ABB RobotStudio station: ABB_Project_EGM_Stream_Single.rspag

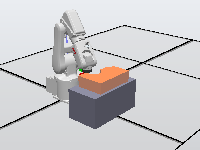
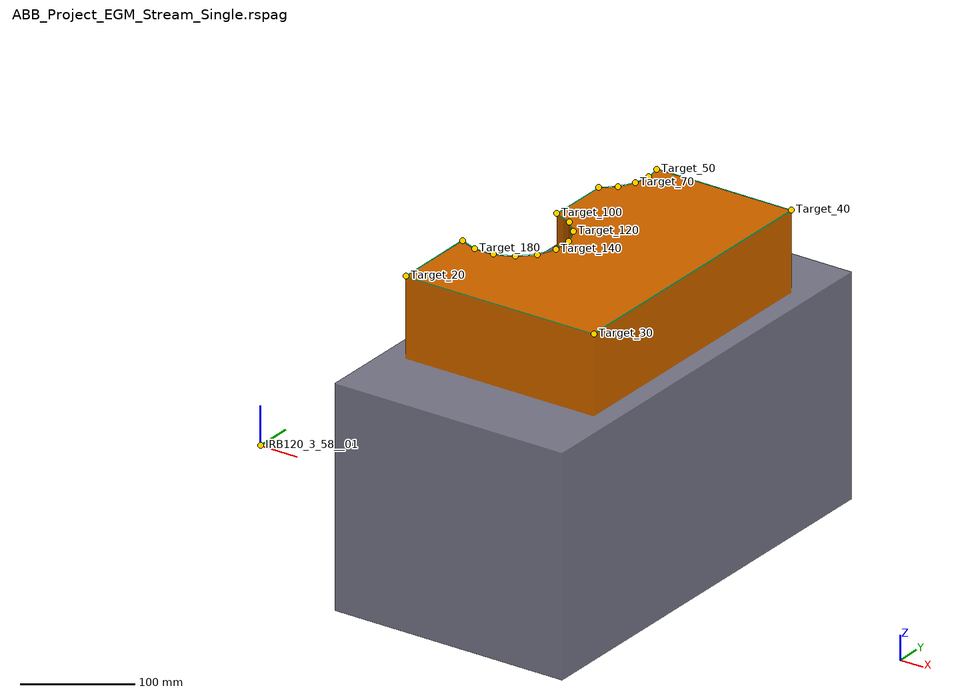
[picture v1: parts stored in the station drawn from their meshes, with robot base, taught points and paths (robot models come from the ABB library and are not in the file)]
--- station ---
Station ABB_Project_EGM_Control (saved by RobotStudio 21.2.9526.0)
Controller Controller2
  mechanical unit ROB_1: IRB120_3_58__01, 6 joints, base frame (0, 0, 0) mm
Layout (positions relative to the parent item):
  - Pad [part] at (250, 150, 200) mm, rotated rx 0 ry 0 rz -90 deg, size 300 x 200 x 100 mm
  - Table [part] at (-40, 0, 0) mm, size 242 x 440 x 220 mm
  - IRB120_3_58__01 [mechanism, from Robots\IRB120_3_58_G_01.rslib] at (0, 0, 0) mm; joint values [-0.2562, 0.0921, 0.7826, 0, 0.6961, -1.827] (rad or m)
Targets, tools, work objects and paths stored in the station and not in the controller backup, written as RAPID:
! task T_ROB1
MODULE Module1
  CONST robtarget Target_10_2:=[[263.321960449,-68.978512397,300],[0,-0.707106781,0.707106781,0],[-1,0,-2,0],[9E+09,9E+09,9E+09,9E+09,9E+09,9E+09]];
  CONST robtarget Target_20_3:=[[263.321960449,-155.446746826,300],[0,-0.707106781,0.707106781,0],[-1,0,-2,0],[9E+09,9E+09,9E+09,9E+09,9E+09,9E+09]];
  CONST robtarget Target_30_3:=[[463.321960449,-155.446746826,300],[0,-0.707106781,0.707106781,0],[-1,0,-2,0],[9E+09,9E+09,9E+09,9E+09,9E+09,9E+09]];
  CONST robtarget Target_40_3:=[[463.321960449,144.553253174,300],[0,-0.707106781,0.707106781,0],[0,0,-1,0],[9E+09,9E+09,9E+09,9E+09,9E+09,9E+09]];
  CONST robtarget Target_50_3:=[[320.448416208,144.553253174,300],[0,-0.707106781,0.707106781,0],[0,0,-1,0],[9E+09,9E+09,9E+09,9E+09,9E+09,9E+09]];
  CONST robtarget Target_60_3:=[[323.349310221,127.995106698,300],[0,-0.707106781,0.707106781,0],[0,0,-1,0],[9E+09,9E+09,9E+09,9E+09,9E+09,9E+09]];
  CONST robtarget Target_70_3:=[[320.59851418,111.411363998,300],[0,-0.707106781,0.707106781,0],[0,0,-1,0],[9E+09,9E+09,9E+09,9E+09,9E+09,9E+09]];
  CONST robtarget Target_80_3:=[[312.506964207,96.676567771,300],[0,-0.707106781,0.707106781,0],[0,0,-1,0],[9E+09,9E+09,9E+09,9E+09,9E+09,9E+09]];
  CONST robtarget Target_90_3:=[[299.98928833,85.456265126,300],[0,-0.707106781,0.707106781,0],[0,0,-1,0],[9E+09,9E+09,9E+09,9E+09,9E+09,9E+09]];
  CONST robtarget Target_100_3:=[[299.98928833,22.036067079,300],[0,-0.707106781,0.707106781,0],[0,0,-1,0],[9E+09,9E+09,9E+09,9E+09,9E+09,9E+09]];
  CONST robtarget Target_110_3:=[[318.046831052,14.718242482,300],[0,-0.707106781,0.707106781,0],[0,0,-1,0],[9E+09,9E+09,9E+09,9E+09,9E+09,9E+09]];
  CONST robtarget Target_120_3:=[[331.936397486,1.05422586,300],[0,-0.707106781,0.707106781,0],[0,0,-1,0],[9E+09,9E+09,9E+09,9E+09,9E+09,9E+09]];
  CONST robtarget Target_130_3:=[[339.548854715,-16.881099643,300],[0,-0.707106781,0.707106781,0],[-1,0,-2,0],[9E+09,9E+09,9E+09,9E+09,9E+09,9E+09]];
  CONST robtarget Target_140_3:=[[339.728249872,-36.364251938,300],[0,-0.707106781,0.707106781,0],[-1,0,-2,0],[9E+09,9E+09,9E+09,9E+09,9E+09,9E+09]];
  CONST robtarget Target_150_3:=[[332.447341773,-54.436711185,300],[0,-0.707106781,0.707106781,0],[-1,0,-2,0],[9E+09,9E+09,9E+09,9E+09,9E+09,9E+09]];
  CONST robtarget Target_160_3:=[[318.811737495,-68.354171512,300],[0,-0.707106781,0.707106781,0],[-1,0,-2,0],[9E+09,9E+09,9E+09,9E+09,9E+09,9E+09]];
  CONST robtarget Target_170_3:=[[300.892005763,-76.003264309,300],[0,-0.707106781,0.707106781,0],[-1,0,-2,0],[9E+09,9E+09,9E+09,9E+09,9E+09,9E+09]];
  CONST robtarget Target_180_3:=[[281.40926075,-76.222473592,300],[0,-0.707106781,0.707106781,0],[-1,0,-2,0],[9E+09,9E+09,9E+09,9E+09,9E+09,9E+09]];
  CONST robtarget Target_190_3:=[[263.321960449,-68.978512397,300],[0,-0.707106781,0.707106781,0],[-1,0,-2,0],[9E+09,9E+09,9E+09,9E+09,9E+09,9E+09]];
  CONST robtarget Target_20_2_3:=[[263.321960449,-155.446746826,300],[0,-0.382683433,0.923879532,0],[-1,0,-1,0],[9E+09,9E+09,9E+09,9E+09,9E+09,9E+09]];
  CONST robtarget Target_30_2_3:=[[463.321960449,-155.446746826,300],[0,0.923879532,-0.382683433,0],[-1,0,-2,0],[9E+09,9E+09,9E+09,9E+09,9E+09,9E+09]];
  CONST robtarget Target_40_2_3:=[[463.321960449,144.553253174,300],[0,0.923879533,0.382683431,0],[0,0,-3,0],[9E+09,9E+09,9E+09,9E+09,9E+09,9E+09]];
  CONST robtarget Target_50_2_3:=[[320.448416208,144.553253174,300],[0,-0.608761429,0.79335334,0],[0,0,-1,0],[9E+09,9E+09,9E+09,9E+09,9E+09,9E+09]];
  CONST robtarget Target_60_2_3:=[[323.349310221,127.995106698,300],[0,-0.5,0.866025404,0],[0,0,-1,0],[9E+09,9E+09,9E+09,9E+09,9E+09,9E+09]];
  CONST robtarget Target_70_2_3:=[[320.59851418,111.411363998,300],[0,-0.382683432,0.923879533,0],[0,0,-1,0],[9E+09,9E+09,9E+09,9E+09,9E+09,9E+09]];
  CONST robtarget Target_80_2_3:=[[312.506964207,96.676567771,300],[0,-0.258819045,0.965925826,0],[0,0,-1,0],[9E+09,9E+09,9E+09,9E+09,9E+09,9E+09]];
  CONST robtarget Target_90_2_3:=[[299.98928833,85.456265126,300],[0,-0.130526192,0.991444861,0],[0,0,0,0],[9E+09,9E+09,9E+09,9E+09,9E+09,9E+09]];
  CONST robtarget Target_100_2_3:=[[299.98928833,22.036067079,300],[0,0.923879533,0.382683432,0],[0,0,1,0],[9E+09,9E+09,9E+09,9E+09,9E+09,9E+09]];
  CONST robtarget Target_110_2_3:=[[318.046831052,14.718242482,300],[0,0.965925826,0.258819045,0],[0,0,1,0],[9E+09,9E+09,9E+09,9E+09,9E+09,9E+09]];
  CONST robtarget Target_120_2_3:=[[331.936397486,1.05422586,300],[0,0.991444861,0.130526192,0],[0,0,1,0],[9E+09,9E+09,9E+09,9E+09,9E+09,9E+09]];
  CONST robtarget Target_130_2_3:=[[339.548854715,-16.881099643,300],[0,1,0,0],[-1,0,1,0],[9E+09,9E+09,9E+09,9E+09,9E+09,9E+09]];
  CONST robtarget Target_140_2_3:=[[339.728249872,-36.364251938,300],[0,0.991444861,-0.130526192,0],[-1,0,2,0],[9E+09,9E+09,9E+09,9E+09,9E+09,9E+09]];
  CONST robtarget Target_150_2_3:=[[332.447341773,-54.436711185,300],[0,0.965925826,-0.258819045,0],[-1,0,2,0],[9E+09,9E+09,9E+09,9E+09,9E+09,9E+09]];
  CONST robtarget Target_160_2_3:=[[318.811737495,-68.354171512,300],[0,0.923879533,-0.382683432,0],[-1,0,2,0],[9E+09,9E+09,9E+09,9E+09,9E+09,9E+09]];
  CONST robtarget Target_170_2_3:=[[300.892005763,-76.003264309,300],[0,0.866025404,-0.5,0],[-1,0,2,0],[9E+09,9E+09,9E+09,9E+09,9E+09,9E+09]];
  CONST robtarget Target_180_2_3:=[[281.40926075,-76.222473592,300],[0,0.79335334,-0.608761429,0],[-1,0,2,0],[9E+09,9E+09,9E+09,9E+09,9E+09,9E+09]];
  CONST robtarget Target_190_2_4:=[[263.321960449,-68.978512397,300],[0,-0.707106781,0.707106781,0],[-1,0,2,0],[9E+09,9E+09,9E+09,9E+09,9E+09,9E+09]];
  CONST robtarget Target_10_2_2_2:=[[263.321960449,-68.978512397,300],[0.092295956,-0.701057385,0.701057385,-0.092295956],[-1,0,-2,0],[9E+09,9E+09,9E+09,9E+09,9E+09,9E+09]];
  CONST robtarget Target_20_2_2_3:=[[263.321960449,-155.446746826,300],[0.092295956,-0.701057385,0.701057385,-0.092295956],[-1,0,-2,0],[9E+09,9E+09,9E+09,9E+09,9E+09,9E+09]];
  CONST robtarget Target_20_2_2_2_2:=[[263.321960449,-155.446746826,300],[0,-0.382683433,0.923879532,0],[-1,0,-1,0],[9E+09,9E+09,9E+09,9E+09,9E+09,9E+09]];
  CONST robtarget Target_30_2_2_3:=[[463.321960449,-155.446746826,300],[0,0.923879532,-0.382683433,0],[-1,0,-2,0],[9E+09,9E+09,9E+09,9E+09,9E+09,9E+09]];
  CONST robtarget Target_30_2_2_2_2:=[[463.321960449,-155.446746826,300],[0.037109679,0.916827972,-0.387892623,-0.087112884],[-1,-1,-2,0],[9E+09,9E+09,9E+09,9E+09,9E+09,9E+09]];
  CONST robtarget Target_40_2_2_3:=[[463.321960449,144.553253174,300],[0.037109679,0.916827972,-0.387892623,-0.087112884],[0,0,-2,0],[9E+09,9E+09,9E+09,9E+09,9E+09,9E+09]];
  CONST robtarget Target_40_2_2_2_2:=[[463.321960449,144.553253174,300],[0,0.923879533,0.382683431,0],[0,0,-3,0],[9E+09,9E+09,9E+09,9E+09,9E+09,9E+09]];
  CONST robtarget Target_60_2_2_2:=[[323.349310221,127.995106698,300],[0,-0.5,0.866025404,0],[0,0,-1,0],[9E+09,9E+09,9E+09,9E+09,9E+09,9E+09]];
  CONST robtarget Target_70_2_2_2:=[[320.59851418,111.411363998,300],[0,-0.382683432,0.923879533,0],[0,0,-1,0],[9E+09,9E+09,9E+09,9E+09,9E+09,9E+09]];
  CONST robtarget Target_80_2_2_2:=[[312.506964207,96.676567771,300],[0,-0.258819045,0.965925826,0],[0,0,-1,0],[9E+09,9E+09,9E+09,9E+09,9E+09,9E+09]];
  CONST robtarget Target_90_2_2_2:=[[299.98928833,85.456265126,300],[0,-0.130526192,0.991444861,0],[0,0,0,0],[9E+09,9E+09,9E+09,9E+09,9E+09,9E+09]];
  CONST robtarget Target_100_2_2_2:=[[299.98928833,22.036067079,300],[0,0.923879533,0.382683432,0],[0,0,1,0],[9E+09,9E+09,9E+09,9E+09,9E+09,9E+09]];
  CONST robtarget Target_110_2_2_2:=[[318.046831052,14.718242482,300],[0,0.965925826,0.258819045,0],[0,0,1,0],[9E+09,9E+09,9E+09,9E+09,9E+09,9E+09]];
  CONST robtarget Target_120_2_2_2:=[[331.936397486,1.05422586,300],[0,0.991444861,0.130526192,0],[0,0,1,0],[9E+09,9E+09,9E+09,9E+09,9E+09,9E+09]];
  CONST robtarget Target_130_2_2_2:=[[339.548854715,-16.881099643,300],[0,1,0,0],[-1,0,1,0],[9E+09,9E+09,9E+09,9E+09,9E+09,9E+09]];
  CONST robtarget Target_140_2_2_2:=[[339.728249872,-36.364251938,300],[0,0.991444861,-0.130526192,0],[-1,0,2,0],[9E+09,9E+09,9E+09,9E+09,9E+09,9E+09]];
  CONST robtarget Target_150_2_2_2:=[[332.447341773,-54.436711185,300],[0,0.965925826,-0.258819045,0],[-1,0,2,0],[9E+09,9E+09,9E+09,9E+09,9E+09,9E+09]];
  CONST robtarget Target_160_2_2_2:=[[318.811737495,-68.354171512,300],[0,0.923879533,-0.382683432,0],[-1,0,2,0],[9E+09,9E+09,9E+09,9E+09,9E+09,9E+09]];
  CONST robtarget Target_170_2_2_2:=[[300.892005763,-76.003264309,300],[0,0.866025404,-0.5,0],[-1,0,2,0],[9E+09,9E+09,9E+09,9E+09,9E+09,9E+09]];
  CONST robtarget Target_180_2_2_2:=[[281.40926075,-76.222473592,300],[0,0.79335334,-0.608761429,0],[-1,0,2,0],[9E+09,9E+09,9E+09,9E+09,9E+09,9E+09]];
  CONST robtarget Target_190_2_3_2:=[[263.321960449,-68.978512397,300],[0,-0.707106781,0.707106781,0],[-1,0,2,0],[9E+09,9E+09,9E+09,9E+09,9E+09,9E+09]];
  PROC Path_Experiment_1_T1()
    MoveL Target_10_2,v40,fine,tool0\WObj:=wobj0;
    MoveL Target_20_3,v40,fine,tool0\WObj:=wobj0;
    MoveL Target_30_3,v40,fine,tool0\WObj:=wobj0;
    MoveL Target_40_3,v40,fine,tool0\WObj:=wobj0;
    MoveL Target_50_3,v40,fine,tool0\WObj:=wobj0;
    MoveL Target_60_3,v40,fine,tool0\WObj:=wobj0;
    MoveL Target_70_3,v40,fine,tool0\WObj:=wobj0;
    MoveL Target_80_3,v40,fine,tool0\WObj:=wobj0;
    MoveL Target_90_3,v40,fine,tool0\WObj:=wobj0;
    MoveL Target_100_3,v40,fine,tool0\WObj:=wobj0;
    MoveL Target_110_3,v40,fine,tool0\WObj:=wobj0;
    MoveL Target_120_3,v40,fine,tool0\WObj:=wobj0;
    MoveL Target_130_3,v40,fine,tool0\WObj:=wobj0;
    MoveL Target_140_3,v40,fine,tool0\WObj:=wobj0;
    MoveL Target_150_3,v40,fine,tool0\WObj:=wobj0;
    MoveL Target_160_3,v40,fine,tool0\WObj:=wobj0;
    MoveL Target_170_3,v40,fine,tool0\WObj:=wobj0;
    MoveL Target_180_3,v40,fine,tool0\WObj:=wobj0;
    MoveL Target_190_3,v40,fine,tool0\WObj:=wobj0;
  ENDPROC
  PROC Path_Experiment_1_T2()
    MoveL Target_10_2,v40,fine,tool0\WObj:=wobj0;
    MoveL Target_20_2_3,v40,fine,tool0\WObj:=wobj0;
    MoveL Target_30_2_3,v40,fine,tool0\WObj:=wobj0;
    MoveL Target_40_2_3,v40,fine,tool0\WObj:=wobj0;
    MoveL Target_50_2_3,v40,fine,tool0\WObj:=wobj0;
    MoveL Target_60_2_3,v40,fine,tool0\WObj:=wobj0;
    MoveL Target_70_2_3,v40,fine,tool0\WObj:=wobj0;
    MoveL Target_80_2_3,v40,fine,tool0\WObj:=wobj0;
    MoveL Target_90_2_3,v40,fine,tool0\WObj:=wobj0;
    MoveL Target_100_2_3,v40,fine,tool0\WObj:=wobj0;
    MoveL Target_110_2_3,v40,fine,tool0\WObj:=wobj0;
    MoveL Target_120_2_3,v40,fine,tool0\WObj:=wobj0;
    MoveL Target_130_2_3,v40,fine,tool0\WObj:=wobj0;
    MoveL Target_140_2_3,v40,fine,tool0\WObj:=wobj0;
    MoveL Target_150_2_3,v40,fine,tool0\WObj:=wobj0;
    MoveL Target_160_2_3,v40,fine,tool0\WObj:=wobj0;
    MoveL Target_170_2_3,v40,fine,tool0\WObj:=wobj0;
    MoveL Target_180_2_3,v40,fine,tool0\WObj:=wobj0;
    MoveL Target_190_2_4,v40,fine,tool0\WObj:=wobj0;
  ENDPROC
  PROC Path_Experiment_1_T3()
    MoveL Target_10_2,v40,z10,tool0\WObj:=wobj0;
    MoveL Target_10_2_2_2,v40,z10,tool0\WObj:=wobj0;
    MoveL Target_20_2_2_3,v40,z10,tool0\WObj:=wobj0;
    MoveL Target_20_2_2_2_2,v40,z10,tool0\WObj:=wobj0;
    MoveL Target_30_2_2_3,v40,z10,tool0\WObj:=wobj0;
    MoveL Target_30_2_2_2_2,v40,z10,tool0\WObj:=wobj0;
    MoveL Target_40_2_2_3,v40,z10,tool0\WObj:=wobj0;
    MoveL Target_40_2_2_2_2,v40,z10,tool0\WObj:=wobj0;
    MoveL Target_50_2_2_2,v40,z10,tool0\WObj:=wobj0;
    MoveL Target_60_2_2_2,v40,z10,tool0\WObj:=wobj0;
    MoveL Target_70_2_2_2,v40,z10,tool0\WObj:=wobj0;
    MoveL Target_80_2_2_2,v40,z10,tool0\WObj:=wobj0;
    MoveL Target_90_2_2_2,v40,z10,tool0\WObj:=wobj0;
    MoveL Target_100_2_2_2,v40,z10,tool0\WObj:=wobj0;
    MoveL Target_110_2_2_2,v40,z10,tool0\WObj:=wobj0;
    MoveL Target_120_2_2_2,v40,z10,tool0\WObj:=wobj0;
    MoveL Target_130_2_2_2,v40,z10,tool0\WObj:=wobj0;
    MoveL Target_140_2_2_2,v40,z10,tool0\WObj:=wobj0;
    MoveL Target_150_2_2_2,v40,z10,tool0\WObj:=wobj0;
    MoveL Target_160_2_2_2,v40,z10,tool0\WObj:=wobj0;
    MoveL Target_170_2_2_2,v40,z10,tool0\WObj:=wobj0;
    MoveL Target_180_2_2_2,v40,z10,tool0\WObj:=wobj0;
    MoveL Target_190_2_3_2,v40,z10,tool0\WObj:=wobj0;
  ENDPROC
ENDMODULE


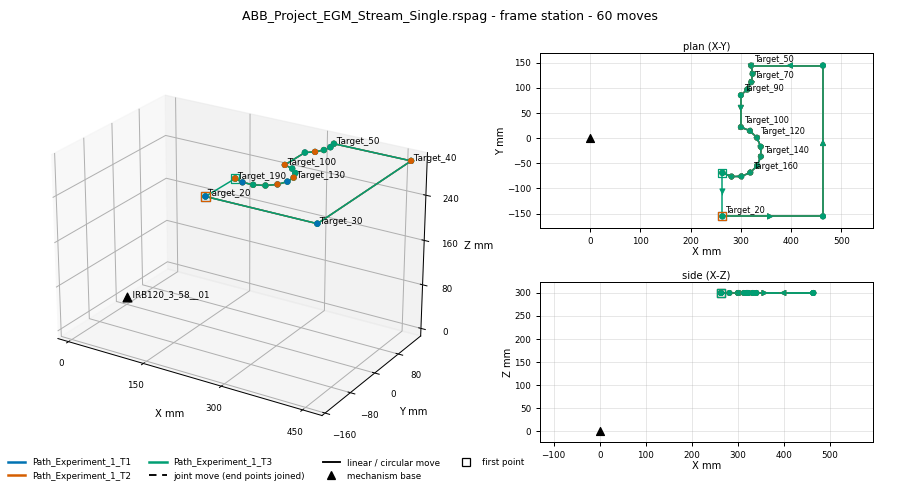
[picture p0: tool path of ABB_Project_EGM_Stream_Single.rspag in frame station, 60 of 60 moves have a stored position in this frame; points joined in program order, loops and branches not executed]
--- Backups/Controller2/RAPID/TASK1/PROGMOD/Module1.mod ---
MODULE Module1
    ! Targets
    CONST robtarget Target_10:=[[263.321960449,-68.978512397,300],[0,-0.707106781,0.707106781,0],[-1,0,-2,0],[9E+09,9E+09,9E+09,9E+09,9E+09,9E+09]];
    CONST robtarget Target_20:=[[263.321960449,-155.446746826,300],[0,-0.707106781,0.707106781,0],[-1,0,-2,0],[9E+09,9E+09,9E+09,9E+09,9E+09,9E+09]];
    CONST robtarget Target_30:=[[463.321960449,-155.446746826,300],[0,-0.707106781,0.707106781,0],[-1,0,-2,0],[9E+09,9E+09,9E+09,9E+09,9E+09,9E+09]];
    CONST robtarget Target_40:=[[463.321960449,144.553253174,300],[0,-0.707106781,0.707106781,0],[0,0,-1,0],[9E+09,9E+09,9E+09,9E+09,9E+09,9E+09]];
    CONST robtarget Target_50:=[[320.448416208,144.553253174,300],[0,-0.707106781,0.707106781,0],[0,0,-1,0],[9E+09,9E+09,9E+09,9E+09,9E+09,9E+09]];
    CONST robtarget Target_60:=[[323.349310221,127.995106698,300],[0,-0.707106781,0.707106781,0],[0,0,-1,0],[9E+09,9E+09,9E+09,9E+09,9E+09,9E+09]];
    CONST robtarget Target_70:=[[320.59851418,111.411363998,300],[0,-0.707106781,0.707106781,0],[0,0,-1,0],[9E+09,9E+09,9E+09,9E+09,9E+09,9E+09]];
    CONST robtarget Target_80:=[[312.506964207,96.676567771,300],[0,-0.707106781,0.707106781,0],[0,0,-1,0],[9E+09,9E+09,9E+09,9E+09,9E+09,9E+09]];
    CONST robtarget Target_90:=[[299.98928833,85.456265126,300],[0,-0.707106781,0.707106781,0],[0,0,-1,0],[9E+09,9E+09,9E+09,9E+09,9E+09,9E+09]];
    CONST robtarget Target_100:=[[299.98928833,22.036067079,300],[0,-0.707106781,0.707106781,0],[0,0,-1,0],[9E+09,9E+09,9E+09,9E+09,9E+09,9E+09]];
    CONST robtarget Target_110:=[[318.046831052,14.718242482,300],[0,-0.707106781,0.707106781,0],[0,0,-1,0],[9E+09,9E+09,9E+09,9E+09,9E+09,9E+09]];
    CONST robtarget Target_120:=[[331.936397486,1.05422586,300],[0,-0.707106781,0.707106781,0],[0,0,-1,0],[9E+09,9E+09,9E+09,9E+09,9E+09,9E+09]];
    CONST robtarget Target_130:=[[339.548854715,-16.881099643,300],[0,-0.707106781,0.707106781,0],[-1,0,-2,0],[9E+09,9E+09,9E+09,9E+09,9E+09,9E+09]];
    CONST robtarget Target_140:=[[339.728249872,-36.364251938,300],[0,-0.707106781,0.707106781,0],[-1,0,-2,0],[9E+09,9E+09,9E+09,9E+09,9E+09,9E+09]];
    CONST robtarget Target_150:=[[332.447341773,-54.436711185,300],[0,-0.707106781,0.707106781,0],[-1,0,-2,0],[9E+09,9E+09,9E+09,9E+09,9E+09,9E+09]];
    CONST robtarget Target_160:=[[318.811737495,-68.354171512,300],[0,-0.707106781,0.707106781,0],[-1,0,-2,0],[9E+09,9E+09,9E+09,9E+09,9E+09,9E+09]];
    CONST robtarget Target_170:=[[300.892005763,-76.003264309,300],[0,-0.707106781,0.707106781,0],[-1,0,-2,0],[9E+09,9E+09,9E+09,9E+09,9E+09,9E+09]];
    CONST robtarget Target_180:=[[281.40926075,-76.222473592,300],[0,-0.707106781,0.707106781,0],[-1,0,-2,0],[9E+09,9E+09,9E+09,9E+09,9E+09,9E+09]];
    CONST robtarget Target_190:=[[263.321960449,-68.978512397,300],[0,-0.707106781,0.707106781,0],[-1,0,-2,0],[9E+09,9E+09,9E+09,9E+09,9E+09,9E+09]];
    CONST robtarget Target_20_2:=[[263.321960449,-155.446746826,300],[0,-0.382683433,0.923879532,0],[-1,0,-1,0],[9E+09,9E+09,9E+09,9E+09,9E+09,9E+09]];
    CONST robtarget Target_30_2:=[[463.321960449,-155.446746826,300],[0,0.923879532,-0.382683433,0],[-1,0,-2,0],[9E+09,9E+09,9E+09,9E+09,9E+09,9E+09]];
    CONST robtarget Target_40_2:=[[463.321960449,144.553253174,300],[0,0.923879533,0.382683431,0],[0,0,-3,0],[9E+09,9E+09,9E+09,9E+09,9E+09,9E+09]];
    CONST robtarget Target_50_2:=[[320.448416208,144.553253174,300],[0,-0.608761429,0.79335334,0],[0,0,-1,0],[9E+09,9E+09,9E+09,9E+09,9E+09,9E+09]];
    CONST robtarget Target_60_2:=[[323.349310221,127.995106698,300],[0,-0.5,0.866025404,0],[0,0,-1,0],[9E+09,9E+09,9E+09,9E+09,9E+09,9E+09]];
    CONST robtarget Target_70_2:=[[320.59851418,111.411363998,300],[0,-0.382683432,0.923879533,0],[0,0,-1,0],[9E+09,9E+09,9E+09,9E+09,9E+09,9E+09]];
    CONST robtarget Target_80_2:=[[312.506964207,96.676567771,300],[0,-0.258819045,0.965925826,0],[0,0,-1,0],[9E+09,9E+09,9E+09,9E+09,9E+09,9E+09]];
    CONST robtarget Target_90_2:=[[299.98928833,85.456265126,300],[0,-0.130526192,0.991444861,0],[0,0,0,0],[9E+09,9E+09,9E+09,9E+09,9E+09,9E+09]];
    CONST robtarget Target_100_2:=[[299.98928833,22.036067079,300],[0,0.923879533,0.382683432,0],[0,0,1,0],[9E+09,9E+09,9E+09,9E+09,9E+09,9E+09]];
    CONST robtarget Target_110_2:=[[318.046831052,14.718242482,300],[0,0.965925826,0.258819045,0],[0,0,1,0],[9E+09,9E+09,9E+09,9E+09,9E+09,9E+09]];
    CONST robtarget Target_120_2:=[[331.936397486,1.05422586,300],[0,0.991444861,0.130526192,0],[0,0,1,0],[9E+09,9E+09,9E+09,9E+09,9E+09,9E+09]];
    CONST robtarget Target_130_2:=[[339.548854715,-16.881099643,300],[0,1,0,0],[-1,0,1,0],[9E+09,9E+09,9E+09,9E+09,9E+09,9E+09]];
    CONST robtarget Target_140_2:=[[339.728249872,-36.364251938,300],[0,0.991444861,-0.130526192,0],[-1,0,2,0],[9E+09,9E+09,9E+09,9E+09,9E+09,9E+09]];
    CONST robtarget Target_150_2:=[[332.447341773,-54.436711185,300],[0,0.965925826,-0.258819045,0],[-1,0,2,0],[9E+09,9E+09,9E+09,9E+09,9E+09,9E+09]];
    CONST robtarget Target_160_2:=[[318.811737495,-68.354171512,300],[0,0.923879533,-0.382683432,0],[-1,0,2,0],[9E+09,9E+09,9E+09,9E+09,9E+09,9E+09]];
    CONST robtarget Target_170_2:=[[300.892005763,-76.003264309,300],[0,0.866025404,-0.5,0],[-1,0,2,0],[9E+09,9E+09,9E+09,9E+09,9E+09,9E+09]];
    CONST robtarget Target_180_2:=[[281.40926075,-76.222473592,300],[0,0.79335334,-0.608761429,0],[-1,0,2,0],[9E+09,9E+09,9E+09,9E+09,9E+09,9E+09]];
    CONST robtarget Target_190_2:=[[263.321960449,-68.978512397,300],[0,-0.707106781,0.707106781,0],[-1,0,2,0],[9E+09,9E+09,9E+09,9E+09,9E+09,9E+09]];
    CONST robtarget Target_10_2_2:=[[263.321960449,-68.978512397,300],[0.092295956,-0.701057385,0.701057385,-0.092295956],[-1,0,-2,0],[9E+09,9E+09,9E+09,9E+09,9E+09,9E+09]];
    CONST robtarget Target_20_2_2:=[[263.321960449,-155.446746826,300],[0.092295956,-0.701057385,0.701057385,-0.092295956],[-1,0,-2,0],[9E+09,9E+09,9E+09,9E+09,9E+09,9E+09]];
    CONST robtarget Target_20_2_2_2:=[[263.321960449,-155.446746826,300],[0,-0.382683433,0.923879532,0],[-1,0,-1,0],[9E+09,9E+09,9E+09,9E+09,9E+09,9E+09]];
    CONST robtarget Target_30_2_2:=[[463.321960449,-155.446746826,300],[0,0.923879532,-0.382683433,0],[-1,0,-2,0],[9E+09,9E+09,9E+09,9E+09,9E+09,9E+09]];
    CONST robtarget Target_30_2_2_2:=[[463.321960449,-155.446746826,300],[0.037109679,0.916827972,-0.387892623,-0.087112884],[-1,-1,-2,0],[9E+09,9E+09,9E+09,9E+09,9E+09,9E+09]];
    CONST robtarget Target_40_2_2:=[[463.321960449,144.553253174,300],[0.037109679,0.916827972,-0.387892623,-0.087112884],[0,0,-2,0],[9E+09,9E+09,9E+09,9E+09,9E+09,9E+09]];
    CONST robtarget Target_40_2_2_2:=[[463.321960449,144.553253174,300],[0,0.923879533,0.382683431,0],[0,0,-3,0],[9E+09,9E+09,9E+09,9E+09,9E+09,9E+09]];
    CONST robtarget Target_50_2_2:=[[320.448416208,144.553253174,300],[0,-0.608761429,0.79335334,0],[0,0,-1,0],[9E+09,9E+09,9E+09,9E+09,9E+09,9E+09]];
    CONST robtarget Target_50_2_2_2:=[[320.448416208,144.553253174,300],[0,-0.608761429,0.79335334,0],[0,-1,-1,0],[9E+09,9E+09,9E+09,9E+09,9E+09,9E+09]];
    CONST robtarget Target_60_2_2:=[[323.349310221,127.995106698,300],[0,-0.5,0.866025404,0],[0,0,-1,0],[9E+09,9E+09,9E+09,9E+09,9E+09,9E+09]];
    CONST robtarget Target_70_2_2:=[[320.59851418,111.411363998,300],[0,-0.382683432,0.923879533,0],[0,0,-1,0],[9E+09,9E+09,9E+09,9E+09,9E+09,9E+09]];
    CONST robtarget Target_80_2_2:=[[312.506964207,96.676567771,300],[0,-0.258819045,0.965925826,0],[0,0,-1,0],[9E+09,9E+09,9E+09,9E+09,9E+09,9E+09]];
    CONST robtarget Target_90_2_2:=[[299.98928833,85.456265126,300],[0,-0.130526192,0.991444861,0],[0,0,0,0],[9E+09,9E+09,9E+09,9E+09,9E+09,9E+09]];
    CONST robtarget Target_100_2_2:=[[299.98928833,22.036067079,300],[0,0.923879533,0.382683432,0],[0,0,1,0],[9E+09,9E+09,9E+09,9E+09,9E+09,9E+09]];
    CONST robtarget Target_110_2_2:=[[318.046831052,14.718242482,300],[0,0.965925826,0.258819045,0],[0,0,1,0],[9E+09,9E+09,9E+09,9E+09,9E+09,9E+09]];
    CONST robtarget Target_120_2_2:=[[331.936397486,1.05422586,300],[0,0.991444861,0.130526192,0],[0,0,1,0],[9E+09,9E+09,9E+09,9E+09,9E+09,9E+09]];
    CONST robtarget Target_130_2_2:=[[339.548854715,-16.881099643,300],[0,1,0,0],[-1,0,1,0],[9E+09,9E+09,9E+09,9E+09,9E+09,9E+09]];
    CONST robtarget Target_140_2_2:=[[339.728249872,-36.364251938,300],[0,0.991444861,-0.130526192,0],[-1,0,2,0],[9E+09,9E+09,9E+09,9E+09,9E+09,9E+09]];
    CONST robtarget Target_150_2_2:=[[332.447341773,-54.436711185,300],[0,0.965925826,-0.258819045,0],[-1,0,2,0],[9E+09,9E+09,9E+09,9E+09,9E+09,9E+09]];
    CONST robtarget Target_160_2_2:=[[318.811737495,-68.354171512,300],[0,0.923879533,-0.382683432,0],[-1,0,2,0],[9E+09,9E+09,9E+09,9E+09,9E+09,9E+09]];
    CONST robtarget Target_170_2_2:=[[300.892005763,-76.003264309,300],[0,0.866025404,-0.5,0],[-1,0,2,0],[9E+09,9E+09,9E+09,9E+09,9E+09,9E+09]];
    CONST robtarget Target_180_2_2:=[[281.40926075,-76.222473592,300],[0,0.79335334,-0.608761429,0],[-1,0,2,0],[9E+09,9E+09,9E+09,9E+09,9E+09,9E+09]];
    CONST robtarget Target_190_2_3:=[[263.321960449,-68.978512397,300],[0,-0.707106781,0.707106781,0],[-1,0,2,0],[9E+09,9E+09,9E+09,9E+09,9E+09,9E+09]];

    ! Home position
    LOCAL CONST robtarget Target_Home:=[[302,0.0,558.0],[0,0,1,0],[-1,0,-1,0],[9E+09,9E+09,9E+09,9E+09,9E+09,9E+09]];
    ! Identifier for the EGM correction
    LOCAL VAR egmident egm_id;

    ! Actual State {Main State-Machine)
    VAR num actual_state := 0;

    ! Initialization Parameters
    CONST num speed_tcp    := 40;
    CONST num speed_orient := 40;
    VAR speeddata speed_value := [speed_tcp,speed_orient,0,0];
    VAR zonedata zone_value   := z0;

    ! Description:                                          !
    ! Simple movements with EGM Streaming Pos. - Main Cycle !
    PROC Main()
        TEST actual_state
            CASE 0:
                ! Register an EGM id
                EGMGetId egm_id;
                ! Setup the EGM communication
                EGMSetupUC ROB_1, egm_id, "default", "ROB_1";
                ! Start the EGM communication session
                EGMStreamStart egm_id \SampleRate:=4;
                actual_state := 1;
            CASE 1:
                ! Move to the starting position
                !MoveJ Target_10,v50,fine,tool0\WObj:=wobj0;

                ! Instructions for multiple movements
                Path_Experiment_1_T1 speed_value, zone_value;
                actual_state := 2;
            CASE 2:
                ! Empty
        ENDTEST

        ! Stop and Release the EGM id
        !EGMStreamStop egm_id;
        !EGMReset egm_id;
    ENDPROC

    PROC Path_Experiment_1_T1(speeddata speed, zonedata zone)
        MoveL Target_20,speed,zone,tool0\WObj:=wobj0;
        MoveL Target_30,speed,zone,tool0\WObj:=wobj0;
        MoveL Target_40,speed,zone,tool0\WObj:=wobj0;
        MoveL Target_50,speed,zone,tool0\WObj:=wobj0;
        MoveL Target_60,speed,zone,tool0\WObj:=wobj0;
        MoveL Target_70,speed,zone,tool0\WObj:=wobj0;
        MoveL Target_80,speed,zone,tool0\WObj:=wobj0;
        MoveL Target_90,speed,zone,tool0\WObj:=wobj0;
        MoveL Target_100,speed,zone,tool0\WObj:=wobj0;
        MoveL Target_110,speed,zone,tool0\WObj:=wobj0;
        MoveL Target_120,speed,zone,tool0\WObj:=wobj0;
        MoveL Target_130,speed,zone,tool0\WObj:=wobj0;
        MoveL Target_140,speed,zone,tool0\WObj:=wobj0;
        MoveL Target_150,speed,zone,tool0\WObj:=wobj0;
        MoveL Target_160,speed,zone,tool0\WObj:=wobj0;
        MoveL Target_170,speed,zone,tool0\WObj:=wobj0;
        MoveL Target_180,speed,zone,tool0\WObj:=wobj0;
        MoveL Target_190,speed,fine,tool0\WObj:=wobj0;
    ENDPROC

    PROC Path_Experiment_1_T2(speeddata speed, zonedata zone)
        MoveL Target_20_2,speed,zone,tool0\WObj:=wobj0;
        MoveL Target_30_2,speed,zone,tool0\WObj:=wobj0;
        MoveL Target_40_2,speed,zone,tool0\WObj:=wobj0;
        MoveL Target_50_2,speed,zone,tool0\WObj:=wobj0;
        MoveL Target_60_2,speed,zone,tool0\WObj:=wobj0;
        MoveL Target_70_2,speed,zone,tool0\WObj:=wobj0;
        MoveL Target_80_2,speed,zone,tool0\WObj:=wobj0;
        MoveL Target_90_2,speed,zone,tool0\WObj:=wobj0;
        MoveL Target_100_2,speed,zone,tool0\WObj:=wobj0;
        MoveL Target_110_2,speed,zone,tool0\WObj:=wobj0;
        MoveL Target_120_2,speed,zone,tool0\WObj:=wobj0;
        MoveL Target_130_2,speed,zone,tool0\WObj:=wobj0;
        MoveL Target_140_2,speed,zone,tool0\WObj:=wobj0;
        MoveL Target_150_2,speed,zone,tool0\WObj:=wobj0;
        MoveL Target_160_2,speed,zone,tool0\WObj:=wobj0;
        MoveL Target_170_2,speed,zone,tool0\WObj:=wobj0;
        MoveL Target_180_2,speed,zone,tool0\WObj:=wobj0;
        MoveL Target_190_2,speed,zone,tool0\WObj:=wobj0;
        MoveJ Target_190,speed,fine,tool0\WObj:=wobj0;
    ENDPROC

    PROC Path_Experiment_1_T3(speeddata speed, zonedata zone)
        MoveL Target_10_2_2,speed,zone,tool0\WObj:=wobj0;
        MoveL Target_20_2_2,speed,zone,tool0\WObj:=wobj0;
        MoveL Target_20_2_2_2,speed,zone,tool0\WObj:=wobj0;
        MoveL Target_30_2_2,speed,zone,tool0\WObj:=wobj0;
        MoveL Target_30_2_2_2,speed,zone,tool0\WObj:=wobj0;
        MoveL Target_40_2_2,speed,zone,tool0\WObj:=wobj0;
        MoveL Target_40_2_2_2,speed,zone,tool0\WObj:=wobj0;
        MoveL Target_50_2_2,speed,zone,tool0\WObj:=wobj0;
        MoveL Target_60_2_2,speed,zone,tool0\WObj:=wobj0;
        MoveL Target_70_2_2,speed,zone,tool0\WObj:=wobj0;
        MoveL Target_80_2_2,speed,zone,tool0\WObj:=wobj0;
        MoveL Target_90_2_2,speed,zone,tool0\WObj:=wobj0;
        MoveL Target_100_2_2,speed,zone,tool0\WObj:=wobj0;
        MoveL Target_110_2_2,speed,zone,tool0\WObj:=wobj0;
        MoveL Target_120_2_2,speed,zone,tool0\WObj:=wobj0;
        MoveL Target_130_2_2,speed,zone,tool0\WObj:=wobj0;
        MoveL Target_140_2_2,speed,zone,tool0\WObj:=wobj0;
        MoveL Target_150_2_2,speed,zone,tool0\WObj:=wobj0;
        MoveL Target_160_2_2,speed,zone,tool0\WObj:=wobj0;
        MoveL Target_170_2_2,speed,zone,tool0\WObj:=wobj0;
        MoveL Target_180_2_2,speed,zone,tool0\WObj:=wobj0;
        MoveL Target_190_2_3,speed,zone,tool0\WObj:=wobj0;
        MoveJ Target_190,speed,fine,tool0\WObj:=wobj0;
    ENDPROC
ENDMODULE
